INTERFACE I_MessageData

PROPERTY DirRoot : POINTER to string(255)
SET
END_SET
END_PROPERTY

PROPERTY ErrorIndex : reference to uint
SET
END_SET
END_PROPERTY

PROPERTY FileRoot : pointer to string(255)
SET
END_SET
END_PROPERTY

PROPERTY LocalTime : pointer to DT
SET
END_SET
END_PROPERTY

PROPERTY MessageIndex : reference to uint
SET
END_SET
END_PROPERTY

PROPERTY MsgList : pointer to ARRAY[1..GVL_MSG_XTS.MAX_MESSAGE] OF st_message
SET
END_SET
END_PROPERTY

END_INTERFACE

(* stored: Version 1.1.0.1
   Itf I_MessageData: Id {d6a51a0f-be9b-4f19-a040-e2a967862d46}
   Property DirRoot: Id {d2c3db40-e38c-40ee-b109-6c5a7e2c3a87}
   Set Set: Id {34f45673-08f4-4fe9-99d9-f068acc0c864}
   Property ErrorIndex: Id {5fcd7088-216e-4ad7-9264-fd86ef87fbb5}
   Set Set: Id {740cad50-812f-4c87-bb6e-7ab469492101}
   Property FileRoot: Id {df55741f-0b3d-4ff9-b733-6ab04ba03107}
   Set Set: Id {4ce6bfbe-bceb-4728-bece-0ef5518f9328}
   Property LocalTime: Id {6c97be70-a955-4256-ad8f-8a2671f9a11f}
   Set Set: Id {b72f632f-9bc7-4d49-8c16-d56bf6157439}
   Property MessageIndex: Id {edad52f5-543e-43d7-8d63-7b31e1fe726b}
   Set Set: Id {8fd909cf-ca31-4492-b638-270491b3dc63}
   Property MsgList: Id {1b3538d6-e6be-4baf-8235-c0ef9eabaa2e}
   Set Set: Id {b49959e4-be6d-4525-95c2-9ccc38048913} *)
